		CASE pMzTool^.P_eObjectType OF
			E_ObjectType.OBJECTTYPE_CartDispenser,
			E_ObjectType.OBJECTTYPE_CartDispStirrer,
			E_ObjectType.OBJECTTYPE_MultiCartHolder,
			E_ObjectType.OBJECTTYPE_PassivPip,
			E_ObjectType.OBJECTTYPE_PiezoPip,
			E_ObjectType.OBJECTTYPE_SolenoidPip,
			E_ObjectType.OBJECTTYPE_PowderPip,
			E_ObjectType.OBJECTTYPE_Extruder,
			E_ObjectType.OBJECTTYPE_TwinExtruder,
			E_ObjectType.OBJECTTYPE_Luer,
			E_ObjectType.OBJECTTYPE_TitrationTool,
			E_ObjectType.OBJECTTYPE_PickPlacePip:
				bMeasureTip := TRUE;
			E_ObjectType.OBJECTTYPE_HybridDispenser:
				//Gemessen wird mit dem MasterTool des Dispensers
				pHybridDispenser := pMzTool;
				pMzTool := pHybridDispenser^.P_pMasterTool;
				bMeasureTip := TRUE;
			E_ObjectType.OBJECTTYPE_StampSupport:	//Vermessung Stamp
				pStampSupport := fbObjectDirectory.M_GetObjPointer(refActionData.nObject);
				IF fbObjectDirectory.M_GetObjType(refActionData.nTarget) = E_ObjectType.OBJECTTYPE_InkStation THEN
					pInkStation := pTarget;
					iTargetZSensor := pInkStation^;
				ELSIF fbObjectDirectory.M_GetObjType(refActionData.nTarget) = E_ObjectType.OBJECTTYPE_StampMagazine THEN
					pStampMagazine := pTarget; 
					iTargetZSensor := pStampMagazine^;
				END_IF
				IF iTargetZSensor.P_bSensor THEN
					M_ExeAction := E_ErrorIdCmd.ERRORID_SensorAlreadySwitched;
					RETURN;
				END_IF
				bMeasureStamp := TRUE;
			E_ObjectType.OBJECTTYPE_ZSensor:	//Vermessung Target
				IF eMeasTipOption = E_MeasureOption.MEAS_OPTION_SlowApproach OR eMeasTipOption = E_MeasureOption.MEAS_OPTION_FastApproach THEN
					bMeasureTarget := TRUE;
				ELSE
					M_ExeAction := E_ErrorIdCmd.ERRORID_InvalidMeasureOption;
					RETURN;				
				END_IF
			ELSE
				M_ExeAction := E_ErrorIdCmd.ERRORID_UnsuitableObject; //Error
				RETURN;				
		END_CASE
		
		
		//Wenn bMeasureTip, dann muss Target ein TipCalibrator sein
		IF bMeasureTip OR bCalibrateTipCalibrator THEN
			IF NOT pTarget^.P_eObjectType = E_ObjectType.OBJECTTYPE_TipCalibrator THEN
				bMeasureTip := FALSE;
				bCalibrateTipCalibrator := FALSE;
				M_ExeAction := E_ErrorIdCmd.ERRORID_UnsuitableTarget;  //Error
				RETURN;
			END_IF
			pTipCalibrator := pTarget;
			bMeasureTipLegacy := pTipCalibrator^.P_bLegacy;
			
			IF pMzTool^.P_pPiece = 0 THEN
				IF pMzTool^.P_eObjectType = E_ObjectType.OBJECTTYPE_PassivPip OR
				   pMzTool^.P_eObjectType = E_ObjectType.OBJECTTYPE_PiezoPip OR
				   pMzTool^.P_eObjectType = E_ObjectType.OBJECTTYPE_SolenoidPip OR
				   pMzTool^.P_eObjectType = E_ObjectType.OBJECTTYPE_Luer THEN
				   rMeasureDistance := 6000;
				ELSIF pMzTool^.P_eObjectType = E_ObjectType.OBJECTTYPE_TitrationTool THEN 
				   rMeasureDistance := 10000;
				ELSE
					M_ExeAction := E_ErrorIdCmd.ERRORID_NoPieceOnTool;
					RETURN;
				END_IF
			ELSE
				IF NOT(pMzTool^.P_pPiece^.P_eObjectType = E_ObjectType.OBJECTTYPE_Nozzle OR
					pMzTool^.P_pPiece^.P_eObjectType = E_ObjectType.OBJECTTYPE_Needle OR
					pMzTool^.P_pPiece^.P_eObjectType = E_ObjectType.OBJECTTYPE_Tip) THEN
					M_ExeAction := E_ErrorIdCmd.ERRORID_InvalidPieceType;
					RETURN;
				ELSE
					rMeasureDistance := pMzTool^.P_pPiece^.P_rMeasureDistance;
				END_IF
			END_IF
		END_IF
		
		M_ExeAction := pMzTool^.M_CheckAction(refActionData, pTarget); //Action mit MzTool ausführbar?
		IF M_ExeAction > 0 THEN
			bMeasureTip := FALSE;
			RETURN;
		END_IF
		
		pHighVoltTray := pTarget^.M_GetFirstParentOfType(E_ObjectType.OBJECTTYPE_HighVoltTray);
		IF pHighVoltTray > 0 THEN
			IF pHighVoltTray^.P_nCurrentVoltage > cHighVoltThreshold THEN //>20 da anloger Eingang etwas rauscht
				M_ExeAction := E_ErrorIdCmd.ERRORID_RiskHighvoltFlashover;
				RETURN;
			END_IF
		END_IF
		
		
	E_Action.ACTION_MoveAllHome:
		;

	E_Action.ACTION_MoveToTarget:
		//Tool ermitteln
		IF fbObjectDirectory.M_ObjIsMzTool(refActionData.nObject) THEN //Gültiges MzTool?
			pMzTool := fbObjectDirectory.M_GetObjPointer(refActionData.nObject);
		ELSE 
			M_ExeAction := E_ErrorIdCmd.ERRORID_UnsuitableObject;  //Error
			RETURN;
		END_IF
		
		IF NOT (fbObjectDirectory.M_GetObjType(refActionData.nObject) = E_ObjectType.OBJECTTYPE_MZHead) THEN
			M_ExeAction := pMzTool^.M_AskSiblingForAction(E_Action.ACTION_MoveToTarget);
			IF M_ExeAction > 0 THEN
				RETURN;
			END_IF
		END_IF
		
		//Falls das Target sich auf dem HighVoltTray befindet und dieses auch angeschalten ist, dann ist ein MoveToTarget nur
		//mit einem MES-Tool möglich
		pTarget := fbObjectDirectory.M_GetObjPointer(refActionData.nTarget);
		IF pTarget = 0 THEN
			M_ExeAction := E_ErrorIdCmd.ERRORID_UnsuitableObject;  //Error
		END_IF
		pHighVoltTray := pTarget^.M_GetFirstParentOfType(E_ObjectType.OBJECTTYPE_HighVoltTray);
		IF pHighVoltTray > 0 THEN
			IF pHighVoltTray^.P_nCurrentVoltage > cHighVoltThreshold AND NOT pMzTool^.P_bIsMESTool THEN
				M_ExeAction := E_ErrorIdCmd.ERRORID_RiskHighvoltFlashover;
				RETURN;
			END_IF
		END_IF
	
		M_ExeAction := fbMoveToTarget.M_SetAndCheckParams(refActionData);

		IF M_ExeAction > 0 THEN
			RETURN;
		END_IF
		
	E_Action.ACTION_OpenCloseFlipTube:
		IF fbObjectDirectory.M_ObjIsMzTool(refActionData.nObject) THEN //Gültiges MzTool?
			pMzTool := fbObjectDirectory.M_GetObjPointer(refActionData.nObject);
		ELSE 
			M_ExeAction := E_ErrorIdCmd.ERRORID_UnsuitableObject;  //Error
			RETURN;
		END_IF
		
		IF fbObjectDirectory.M_ObjIsTarget(refActionData.nTarget) THEN //Gültiges Target?
			pTarget := fbObjectDirectory.M_GetObjPointer(refActionData.nTarget);
			IF pTarget^.P_eObjectType = E_ObjectType.OBJECTTYPE_FlipTubeRack THEN //Target ein FlipTubeRack?
				pFlipTubeRack := pTarget;
				pPieceSlot := pFlipTubeRack^.M_GetSlot(DINT_TO_UINT(refActionData.aParams[1]));
			ELSE
				M_ExeAction := E_ErrorIdCmd.ERRORID_UnsuitableTarget;  //Error	
			END_IF
		ELSE
			M_ExeAction := E_ErrorIdCmd.ERRORID_UnsuitableTarget;  //Error
			RETURN;
		END_IF
		
		M_ExeAction := pMzTool^.M_CheckAction(refActionData, pTarget); //Ausführbar mit Target?
		IF M_ExeAction > 0 THEN
			RETURN;
		END_IF
		
		M_ExeAction := pTarget^.M_CheckAction(refActionData, pMzTool); //Ausführbar mit MzTool?
		IF M_ExeAction > 0 THEN
			RETURN;
		END_IF
		bOpen := NOT DINT_TO_BOOL(refActionData.aParams[2]); //Öffen
		
	E_Action.ACTION_StampDemolding:
		IF fbObjectDirectory.M_GetObjType(refActionData.nObject) <> E_ObjectType.OBJECTTYPE_StampSupport THEN //Gültiges MzTool?
			M_ExeAction := E_ErrorIdCmd.ERRORID_UnsuitableObject;
			RETURN;
		END_IF
		pMzTool := fbObjectDirectory.M_GetObjPointer(refActionData.nObject);
		pStampSupport := pMzTool;

		M_ExeAction := pStampSupport^.M_CheckAction(refActionData,0);
		IF M_ExeAction > 0 THEN
			RETURN;
		END_IF
 
		nDistance1 := refActionData.aParams[1];
		nSpeed1 := refActionData.aParams[2];
		nPressure1 := DINT_TO_INT(refActionData.aParams[3]);
		nPressure2 := DINT_TO_INT(refActionData.aParams[4]);
		nPeriode := refActionData.aParams[5];
		nDutycycle := refActionData.aParams[6];
		
	E_Action.ACTION_StampInking:
		IF fbObjectDirectory.M_GetObjType(refActionData.nObject) <> E_ObjectType.OBJECTTYPE_StampSupport THEN //Gültiges MzTool?
			M_ExeAction := E_ErrorIdCmd.ERRORID_UnsuitableObject;
			RETURN;
		END_IF
		
		//Inking kann an einem Punkt oder an der InkStation stattfinden
		IF fbObjectDirectory.M_GetObjType(refActionData.nTarget) = E_ObjectType.OBJECTTYPE_InkStation THEN
			pInkStation := fbObjectDirectory.M_GetObjPointer(refActionData.nTarget);
		ELSIF fbObjectDirectory.M_GetObjType(refActionData.nTarget) = E_ObjectType.OBJECTTYPE_Point THEN
			pInkStation := 0;
		ELSE
			M_ExeAction := E_ErrorIdCmd.ERRORID_UnsuitableTarget;
			RETURN;
		END_IF
		
		//Wozu brauchen wir hier das Target?
		pTarget := fbObjectDirectory.M_GetObjPointer(refActionData.nTarget);
		pStampSupport := fbObjectDirectory.M_GetObjPointer(refActionData.nObject);
		
		M_ExeAction := pStampSupport^.M_CheckAction(refActionData,pTarget);
		IF M_ExeAction > 0 THEN
			RETURN;
		END_IF
		
		nDistance1 := refActionData.aParams[1];
		nPressure1 := DINT_TO_INT(refActionData.aParams[2]);
		nTime := DINT_TO_DWORD(refActionData.aParams[3]);
		
	E_Action.ACTION_TeachTarget:
		//Object gültig?
		IF NOT fbObjectDirectory.M_ObjIsMzTool(refActionData.nObject) THEN
			M_ExeAction := E_ErrorIdCmd.ERRORID_UnsuitableObject;  //Error
			RETURN;
		END_IF
		
		IF fbObjectDirectory.M_ObjIsTarget(refActionData.nTarget) THEN
			pTarget := fbObjectDirectory.M_GetObjPointer(refActionData.nTarget);
			IF pTarget > 0 THEN
				M_ExeAction := pTarget^.M_CheckAction(refActionData, pMzTool);
				IF M_ExeAction > 0 THEN
					RETURN;
				END_IF
			ELSE
				M_ExeAction := E_ErrorIdCmd.ERRORID_UnsuitableTarget;  //Error
				RETURN;
			END_IF
		ELSE
			M_ExeAction := E_ErrorIdCmd.ERRORID_UnsuitableTarget;  //Error
			RETURN;
		END_IF
		//Target gültig? (derzeit nur Mtp impl.)
		
		//Hier macht es Sinn, beim Target selber zu fragen, ob es sich einteachen lässt
		
		(*IF fbObjectDirectory.M_GetObjType(refActionData.nTarget) = E_ObjectType.OBJECTTYPE_Mtp THEN
			pMtp := aI_Object[refActionData.nTarget].P_pObject;
		ELSIF fbObjectDirectory.M_GetObjType(refActionData.nTarget) = E_ObjectType.OBJECTTYPE_Point THEN
			;
		ELSIF fbObjectDirectory.M_GetObjType(refActionData.nTarget) = E_ObjectType.OBJECTTYPE_Stroboscope THEN
			;
		ELSE
			M_ExeAction := E_ErrorIdCmd.ERRORID_InvalidTarget;  //Error
			RETURN;
		END_IF*)
		
		pMzTool := fbObjectDirectory.M_GetObjPointer(refActionData.nObject);
		pTarget := fbObjectDirectory.M_GetObjPointer(refActionData.nTarget);
		IF pTarget^.P_eObjectType = E_ObjectType.OBJECTTYPE_Mtp THEN
			pMtp := pTarget;
		END_IF
		eTargetRef := DINT_TO_USINT(refActionData.aParams[1]);
		nSpecPointSlotNr := DINT_TO_UINT(refActionData.aParams[2]);
		nZOffset1 := refActionData.aParams[3];
		//refActionData.aParams[4] ist Reserve
		eTeachOption := DINT_TO_USINT(refActionData.aParams[5]);
		
		pHighVoltTray := pTarget^.M_GetFirstParentOfType(E_ObjectType.OBJECTTYPE_HighVoltTray);
		IF pHighVoltTray > 0 THEN
			IF pHighVoltTray^.P_nCurrentVoltage > cHighVoltThreshold THEN
				M_ExeAction := E_ErrorIdCmd.ERRORID_RiskHighvoltFlashover;
				RETURN;
			END_IF
		END_IF
		
	E_Action.ACTION_TeachTool:
		IF NOT fbObjectDirectory.M_ObjIsMzTool(refActionData.nObject) THEN
			M_ExeAction := E_ErrorIdCmd.ERRORID_UnsuitableObject;  //Error
			RETURN;
		END_IF
		//Target gültig?
		IF NOT fbObjectDirectory.M_ObjIsTarget(refActionData.nTarget) THEN
			M_ExeAction := E_ErrorIdCmd.ERRORID_UnsuitableTarget;  //Error
			RETURN;
		END_IF
		pMzTool := fbObjectDirectory.M_GetObjPointer(refActionData.nObject);
		pTarget := fbObjectDirectory.M_GetObjPointer(refActionData.nTarget);
		eTargetRef := DINT_TO_USINT(refActionData.aParams[1]);
		nCol := DINT_TO_USINT(refActionData.aParams[2]);
		nRow := DINT_TO_USINT(refActionData.aParams[2]);
		nZOffset1 := refActionData.aParams[4];

		pHighVoltTray := pTarget^.M_GetFirstParentOfType(E_ObjectType.OBJECTTYPE_HighVoltTray);
		IF pHighVoltTray > 0 THEN
			IF pHighVoltTray^.P_nCurrentVoltage > cHighVoltThreshold THEN
				M_ExeAction := E_ErrorIdCmd.ERRORID_RiskHighvoltFlashover;
				RETURN;
			END_IF
		END_IF

	E_Action.ACTION_TransferGas:
		//Beteiligte Luers checken
		IF NOT fbObjectDirectory.M_GetObjType(refActionData.nObject) = E_ObjectType.OBJECTTYPE_Luer THEN
			M_ExeAction := E_ErrorIdCmd.ERRORID_UnsuitableObject;  //Error
			RETURN;
		END_IF

		IF NOT fbObjectDirectory.M_GetObjType(refActionData.nTarget) = E_ObjectType.OBJECTTYPE_Luer THEN
			M_ExeAction := E_ErrorIdCmd.ERRORID_UnsuitableObject;  //Error
			RETURN;
		END_IF
		pLuer := fbObjectDirectory.M_GetObjPointer(refActionData.nObject);
		pLuer2 := fbObjectDirectory.M_GetObjPointer(refActionData.nTarget);
		nPressure1 := DINT_TO_INT(refActionData.aParams[1]);
		nTime := DINT_TO_DWORD(refActionData.aParams[2]);
		
	E_Action.ACTION_TransferLiquid:
		//Beteiligte Luers checken
		IF NOT fbObjectDirectory.M_GetObjType(refActionData.nObject) = E_ObjectType.OBJECTTYPE_Luer THEN
			M_ExeAction := E_ErrorIdCmd.ERRORID_UnsuitableObject;  //Error
			RETURN;
		END_IF

		IF NOT fbObjectDirectory.M_GetObjType(refActionData.nTarget) = E_ObjectType.OBJECTTYPE_Luer THEN
			M_ExeAction := E_ErrorIdCmd.ERRORID_UnsuitableTarget;  //Error
			RETURN;
		END_IF
		pLuer := fbObjectDirectory.M_GetObjPointer(refActionData.nObject);
		pLuer2 := fbObjectDirectory.M_GetObjPointer(refActionData.nTarget);
		pDiluter1 := pLuer^.P_pDiluter;
		pDiluter2 := pLuer2^.P_pDiluter;
		
		nQuantity1 := refActionData.aParams[1];
		nFlow1 := refActionData.aParams[2];
		nQuantity2 := refActionData.aParams[3];
		nQuantity3 := refActionData.aParams[4];
		
	E_Action.ACTION_TransferTray:
		//Hier schon Bedingungen abfragen.
		IF fbObjectDirectory.M_GetObjType(refActionData.nObject) = E_ObjectType.OBJECTTYPE_TrayTransporter THEN
			pTrayTransporter := fbObjectDirectory.M_GetObjPointer(refActionData.nObject);
		ELSE
			M_ExeAction := E_ErrorIdCmd.ERRORID_UnsuitableObject;  //Error
			RETURN;
		END_IF
 
		eTransferTrayCtrl :=  DINT_TO_USINT(refActionData.aParams[1]);

	E_Action.ACTION_WashTool:
		IF fbObjectDirectory.M_ObjIsMzTool(refActionData.nObject) THEN //Gültiges MzTool?
			pMzTool := fbObjectDirectory.M_GetObjPointer(refActionData.nObject);
		ELSE 
			M_ExeAction := E_ErrorIdCmd.ERRORID_UnsuitableObject;  //Error
			RETURN;
		END_IF	
		
		IF fbObjectDirectory.M_GetObjType(refActionData.nTarget) <> E_ObjectType.OBJECTTYPE_WashStation THEN //gültiges Target?
			M_ExeAction := E_ErrorIdCmd.ERRORID_UnsuitableTarget;
			RETURN;
		ELSE
			pTarget := fbObjectDirectory.M_GetObjPointer(refActionData.nTarget);
			pWashStation := pTarget;
		END_IF
		
		//Kann Tool Action ausführen?
		M_ExeAction := pMzTool^.M_CheckAction(refActionData, pTarget);
		IF M_ExeAction > 0 THEN
			RETURN;
		END_IF
		
		//Kann WashStation Action ausführen?
		M_ExeAction := pWashStation^.M_CheckAction(refActionData, pMzTool);
		IF M_ExeAction > 0 THEN
			RETURN;
		END_IF
		
		nSpecPointSlotNr := DINT_TO_UINT(refActionData.aParams[1]);
		//RinseChannel aus WashStation holen
		nRinseChannel := pWashStation^.M_GetRinseChannel(UINT_TO_USINT(nSpecPointSlotNr));
		eWashMode := DINT_TO_USINT(refActionData.aParams[2]);
		//passt WashMode zu RinseChannel?
		IF (eWashMode = E_WashMode.MODE_WashInOutside) OR (eWashMode = E_WashMode.MODE_WashOutside) THEN
			IF nRinseChannel = 0 THEN
				M_ExeAction := E_ErrorIdCmd.ERRORID_InvalidRinseChannel;
				RETURN;
			END_IF
		END_IF
		
		nQuantity1 := refActionData.aParams[3];
		nFlow1 := refActionData.aParams[4];
		nTime := DINT_TO_DWORD(refActionData.aParams[5]);
		nDilInputNr := refActionData.aParams[6];

 	ELSE
		M_ExeAction := E_ErrorIdCmd.ERRORID_InvalidAction; //Error		
END_CASE
bBusy := TRUE;
eCurrentAction := refActionData.eAction;
eCurrentState := E_MachineState.MACHINESTATE_Active;
END_METHOD

METHOD M_Pause
VAR_INPUT
END_VAR
//derzeit wird nur DispenseTest in Pause versetzt
IF eCurrentState = E_MachineState.MACHINESTATE_Active THEN
	IF eCurrentAction = E_Action.ACTION_DispenseTest THEN
		eCurrentState := E_MachineState.MACHINESTATE_PauseRequest;
	END_IF
END_IF
END_METHOD

METHOD M_Reset
VAR_INPUT
END_VAR
VAR
END_VAR
IF eCurrentState = E_MachineState.MACHINESTATE_Error THEN
	bBusy := TRUE;
	eCurrentState := E_MachineState.MACHINESTATE_Reset;
END_IF
END_METHOD

METHOD M_Stop
VAR_INPUT
END_VAR
IF eCurrentState = E_MachineState.MACHINESTATE_Active OR 
	eCurrentState = E_MachineState.MACHINESTATE_PauseRequest OR
	eCurrentState = E_MachineState.MACHINESTATE_Pause THEN
	
	bStop := TRUE;
END_IF
END_METHOD

METHOD M_StopAction
VAR_INPUT
	eAction : E_Action;
END_VAR
IF eCurrentAction = eAction THEN
	M_Stop();
END_IF
END_METHOD

PROPERTY P_bLastActionResult : BOOL
GET
P_bLastActionResult := bLastActionResult;
END_GET
SET
bLastActionResult := P_bLastActionResult;
END_SET
END_PROPERTY

PROPERTY P_bPauseRequestIntern : BOOL
GET
P_bPauseRequestIntern := bPauseRequestIntern;
END_GET
SET
bPauseRequestIntern := P_bPauseRequestIntern;
END_SET
END_PROPERTY

PROPERTY P_nDispenseTrials : DINT
GET
P_nDispenseTrials := nDispenseTrials;
END_GET
SET
nDispenseTrials := P_nDispenseTrials;
END_SET
END_PROPERTY

PROPERTY P_nLastActionResult : DINT
GET
P_nLastActionResult := nLastActionResult;
END_GET
SET
nLastActionResult := P_nLastActionResult;
END_SET
END_PROPERTY

END_FUNCTION_BLOCK

// ---- Hardware/MultiZ/FB_ZM_ReadZSensorID.TcPOU
FUNCTION_BLOCK FB_ZM_ReadZSensorID
VAR_INPUT
	bExecute		: BOOL;
	pFbZAxisRef		: POINTER TO FB_ZAxisRef;
END_VAR
VAR_OUTPUT
	bBusy			: BOOL;
	bCommandAborted	: BOOL;
	bError			: BOOL;
	nErrorID		: ERRORID;	
END_VAR
VAR
	nState				: USINT;
	timeOut				: TON;
	fbSdoRead			: FB_SDO_READ;
END_VAR

//Die Id (eigentlich der Offset) wird ausgelesen, indem eine kurze Vermessung mit 100µm Distanz gestartet wird.
//Als Ergebnis bringt die Achse einen der 3 folgenden Fehler:
//1. No_Z-Limit -> kein ZSensor (Id wurde nicht ausgelesen)
//2. Z_Limit_Fail -> ZSensor betätigt (Id wurde ausgelesen)
//3. Z_Limit_not_found -> (Id wurde ausgelesen)

IF bExecute THEN
	IF pFbZAxisRef = 0 THEN
		nErrorId := E_ErrorIdMultiZ.ERRORID_InvalidZChannel;
		bBusy := FALSE;
		bError := TRUE;
		nState := 99;
		RETURN;
	END_IF

	//Wenn durch anderen FB Achse gestoppt, dann abbrechen
	IF pFbZAxisRef^.stStatus.bCmdAborted THEN //Muss noch irgendwo gesetzt werden!!!!
		bCommandAborted := TRUE;
		bBusy := FALSE;
	END_IF
	
	timeOut();
	IF timeOut.Q THEN
		bBusy := FALSE;
		bError := TRUE;
		nState := 99;
		RETURN;
	END_IF

	CASE nState OF
		0: 	//Nur folgende Tools können ZSensor aufnehmen
			bBusy := TRUE;
			IF NOT (pFbZAxisRef^.eFixedToolType = E_MzToolType.TOOL_TYPE_PiezoPip OR 
					pFbZAxisRef^.eFixedToolType = E_MzToolType.TOOL_TYPE_PiezoSingle OR 
					pFbZAxisRef^.eFixedToolType = E_MzToolType.TOOL_TYPE_SyringeExtruder) THEN
				nErrorID := E_ErrorIdCmd.ERRORID_ConfigErrorZSensor;
				bBusy := FALSE;
				bError := TRUE;
				nState := 99;
				RETURN;
			END_IF
			
			pFbZAxisRef^.stStatus.bIsMoving := TRUE;
			pFbZAxisRef^.stStatus.bHasJob := TRUE;
        	//Geschwindigkeit setzen
			pFbZAxisRef^.stOutput.nVelo := REAL_TO_DINT(pFbZAxisRef^.P_rMaxSpeed);
			//Aktuelle Position ? Wenn ganz unten steht, dann 200µ nach oben fahren
			IF (pFbZAxisRef^.P_rCurrentPos - 100.0) < pFbZAxisRef^.P_rMinPos THEN
				//200µm nach oben fahren
				pFbZAxisRef^.stOutput.nMode := 1; //normaler Positioniermodus
				pFbZAxisRef^.P_rAbsTargetPos := pFbZAxisRef^.P_rMinPos + 200.0;
				pFbZAxisRef^.stOutput.nCtrl := 1;
				nState := 1;
			ELSE
				nState := 3;
			END_IF
			
		1:	//SetpointAcknowledge?
			IF pFbZAxisRef^.stInput.nStatus.1 THEN
				pFbZAxisRef^.stOutput.nCtrl.0 := FALSE;	//Fahrauftrag zurücksetzen
				timeOut(IN:= FALSE);
				nState := 2;
			ELSE
				timeOut(IN:= TRUE, PT:=T#1000MS);	//Timer für Timeout starten
			END_IF
			
		2:  //TargetReached?
			IF pFbZAxisRef^.stInput.nStatus.0 THEN
				timeOut(IN:= FALSE);
				nState := 3;
			ELSE
				timeOut(IN:= TRUE, PT:= T#1000MS);	//Timer für Timeout starten
			END_IF			
			
		3:	//100µm nach unten im Messmodus fahren -> sollte in jedem Fall einen Fehler erzeugen
			//Hier muss kurzzeitig verhindert werden, dass dieser Fehler in Action "A_Monitor" von
			//FB_MultiZRef abgefangen wird
			pFbZAxisRef^.stOutput.nMode := 5; //normaler Messmodus
			pFbZAxisRef^.stOutput.nTrgtPos := 100;
			pFbZAxisRef^.bIngoreError := TRUE;
			nState := 4;
			
		4:	pFbZAxisRef^.stOutput.nCtrl := 1;
			nState := 5;
			
		5:	//SetpointAcknowledge?
			IF pFbZAxisRef^.stInput.nStatus.1 THEN
				pFbZAxisRef^.stOutput.nCtrl.0 := FALSE;	//Fahrauftrag zurücksetzen
				timeOut(IN:= FALSE);
				timeOut(IN:= TRUE, PT:= T#1S);
				nState := 6;
			ELSE
				timeOut(IN:= TRUE, PT:=T#1000MS);	//Timer für Timeout starten
			END_IF

		6:	//Hier sollte jetzt ein Fehler kommen
			IF pFbZAxisRef^.stInput.nStatus.3 AND pFbZAxisRef^.stInput.nError > 0 THEN
				pFbZAxisRef^.stOutput.nMode := 0; //Mode muss zum Zurücksetzen des Fehlers auf 0 sein
				timeOut(IN:= FALSE);
				nErrorID := pFbZAxisRef^.stInput.nError;
				IF nErrorID = 19 OR nErrorID = 20 THEN
					//weiter zu Offset auslesen und Error zurücksetzen
					fbSdoRead(sADSNetID:= pFbZAxisRef^.pMultiZRef^.P_sAdsNetId,	nPortNr:= pFbZAxisRef^.pMultiZRef^.P_nAdsPort,
							nIndex:= cZSensOffset.nIndex, nSubIndex:= pFbZAxisRef^.nChannel, nDataLength:= cZSensOffset.nLength, bExecute:= TRUE);					
					nState := 7;
				ELSE
					nErrorID := F_MultiZError_TO_ErrorId(pFbZAxisRef^.stInput.nError);
					bBusy := FALSE;
					bError := TRUE;
					RETURN;					
				END_IF
			END_IF
			
		7:	//Warten bis ZOffset ausgelesen
			fbSdoRead();
			IF NOT fbSdoRead.bBusy THEN
				IF fbSdoRead.bError THEN
					nErrorID := fbSdoRead.nAdsErrorId;
					bError := TRUE;
					nState := 99;
				ELSE
					nState := 8;
					pFbZAxisRef^.stOutput.nCtrl := 8;	//Error zurücksetzen
					pFbZAxisRef^.P_nZSensorID := fbSdoRead.nData;
				END_IF
				fbSdoRead(bExecute:= FALSE);
			END_IF
			
		8:	IF NOT pFbZAxisRef^.stInput.nStatus.3 AND pFbZAxisRef^.stInput.nError = 0 THEN
				pFbZAxisRef^.stOutput.nCtrl := 0;
				bBusy := FALSE;				
			END_IF
	END_CASE
ELSE
	bBusy := FALSE;
	nState := 0;
	bError := FALSE;
	nErrorID := 0;
	timeOut(IN:=FALSE);
	pFbZAxisRef^.stStatus.bCmdAborted := FALSE;
	pFbZAxisRef^.stOutput.nMode := 0;
	pFbZAxisRef^.stStatus.bHasJob := FALSE;
	pFbZAxisRef^.stStatus.bIsMoving := FALSE;
	pFbZAxisRef^.bIngoreError := FALSE;
END_IF

END_FUNCTION_BLOCK

// ---- Actions/FB_MeasTip.TcPOU
FUNCTION_BLOCK FB_MeasTip
VAR_INPUT
	bExecute 		: BOOL;
	pMzTool			: POINTER TO FB_MzBase;
	pTipCalibrator	: POINTER TO FB_TipCalibrator;
	nDirection 		: USINT;	//1: X, 2: Y, 3: Z
	nZFeedStart		: DINT;		//Anfangsschrittweite in Z (µm)
	nZFeedEnde		: DINT;		//Endschrittweite in Z (µm)
	nZFeedMax		: DINT;
	stStartPos		: ST_3DPoint;
	stEndPos		: ST_3DPoint;
	stTempPoint		: ST_3DPoint;
END_VAR
VAR_OUTPUT
	bBusy		: BOOL;
	bError		: BOOL;
	nErrorId	: ERRORID;
	stProbePos	: ST_3DPoint;
END_VAR
VAR
	stError				: ST_Error;
	pXDrive				: POINTER TO FB_XYDriveBase;
	pYDrive				: POINTER TO FB_XYDriveBase;
	nState				: USINT;
	stCurrentPos		: ST_3DPoint;
	stCalibPoint		: ST_3DPoint;
	stPassIntersect		: ST_3DPoint;	
	stActionData		: ST_ActionData;
	rCapturedPos1		: REAL;
	rCapturedPos2		: REAL;
	nStateA_ProbeX		: USINT;
	nStateA_ProbeY		: USINT;
	bSingleProbe		: BOOL;
	bDirPositive		: BOOL;
	nStartPos			: DINT;
	nEndPos				: DINT;
	bBeginStartPos		: BOOL;
	nProbeSpeed			: DINT := 20000;
	bProbeSuccess		: BOOL;
	nProbeErrorId		: UINT;
	bProbePositiveOK	: BOOL;
	bProbeNegativeOK	: BOOL;
	bProbeMissingTouch	: BOOL;
	bProbeFlag			: BOOL;
	bTouchProbe			: BOOL;
	nProbeCount			: USINT;
	nZFeed				: DINT;
	nZFeedSum			: DINT;
	bMaxFeedAchieved	: BOOL;
END_VAR

IF bExecute THEN
	IF nDirection = 1 THEN	//X
		A_MeasureX();
	ELSIF nDirection = 2 THEN //Y
		A_MeasureY();
	ELSIF nDirection = 3 THEN	//Z
		A_MeasureZ();
	END_IF
ELSE
	bError := FALSE;
	nErrorId := 0;
	nState := 0;
	nStateA_ProbeX := 0;
	nStateA_ProbeY := 0;
END_IF

ACTION A_MeasureX:
IF pMzTool^.P_bError THEN
	nState := 99;
	bError := TRUE;
	stError := pMzTool^.P_stError;
	nErrorId := stError.ErrorId; 
END_IF

CASE nState OF
	0:	
		nStartPos := REAL_TO_DINT(stStartPos.X);
		nEndPos := REAL_TO_DINT(stEndPos.X);
		bBusy := TRUE;
		bBeginStartPos := TRUE;
		bSingleProbe := FALSE;
		nState := 1;

	1:	//XProbe
		A_ProbeX();
		IF nStateA_ProbeX = 80 THEN
			nStateA_ProbeX := 0;
			IF bProbeSuccess AND bProbePositiveOK AND bProbeNegativeOK THEN
				//Checken, ob beide Probe-Positionen nicht zu weit voneinander abweichen (max5mm)
				IF ABS(rCapturedPos1 - rCapturedPos2) > 20000 THEN
					bError := TRUE;
					nErrorId := E_ErrorIdCmd.ERRORID_MeasureTouchProbeFail;
					bBusy := FALSE;
					RETURN;	
				END_IF				
				stTempPoint.X := (rCapturedPos1 + rCapturedPos2) / 2;
				stTempPoint :=  pMzTool^.M_RawPosToRealPos(stTempPoint);
				stProbePos.X := stTempPoint.X;
				bBusy := FALSE;	
			END_IF
		ELSIF nStateA_ProbeX = 99 THEN
			nStateA_ProbeX := 0;
			bBusy := FALSE;
			bError := TRUE;
			nErrorId := nProbeErrorId;
		END_IF
		
	70:	//Abbrechen
		IF nStateA_ProbeX > 0 THEN
			nStateA_ProbeX := 70;
			A_ProbeX();
			nState := 71;
		END_IF
		
	71:	
		A_ProbeX();
		IF nStateA_ProbeX >= 80 THEN
			IF nStateA_ProbeX >= 99 THEN
				nErrorId := nProbeErrorId;
				bError := TRUE;
			END_IF
			nStateA_ProbeX := 0;
			bBusy := FALSE;
		END_IF
END_CASE
END_ACTION

ACTION A_MeasureY:
IF pMzTool^.P_bError THEN
	nState := 90;
	bError := TRUE;
	stError := pMzTool^.P_stError;
	nErrorId := stError.ErrorId; 
END_IF

CASE nState OF
	0:	
		nStartPos := REAL_TO_DINT(stStartPos.Y);
		nEndPos := REAL_TO_DINT(stEndPos.Y);
		bBusy := TRUE;
		bBeginStartPos := FALSE;
		bSingleProbe := FALSE;
		nState := 1;

	1:	//YProbe
		A_ProbeY();
		IF nStateA_ProbeY = 80 THEN
			nStateA_ProbeY := 0;
			IF bProbeSuccess AND bProbePositiveOK AND bProbeNegativeOK THEN
				//Checken, ob beide Probe-Positionen nicht zu weit voneinander abweichen (max5mm)
				IF ABS(rCapturedPos1 - rCapturedPos2) > 20000 THEN
					bError := TRUE;
					nErrorId := E_ErrorIdCmd.ERRORID_MeasureTouchProbeFail;
					bBusy := FALSE;
					RETURN;	
				END_IF
				stTempPoint.Y := (rCapturedPos1 + rCapturedPos2) / 2;
				stTempPoint :=  pMzTool^.M_RawPosToRealPos(stTempPoint);
				stProbePos.Y := stTempPoint.Y;
				bBusy := FALSE;	
			END_IF
		ELSIF nStateA_ProbeY = 99 THEN
			nStateA_ProbeY := 0;
			bBusy := FALSE;
			bError := TRUE;
			nErrorId := nProbeErrorId;
		END_IF
		
	70:	//Abbrechen
		IF nStateA_ProbeY > 0 THEN
			nStateA_ProbeY := 70;
			A_ProbeY();
			nState := 71;
		END_IF
		
	71:	
		A_ProbeY();
		IF nStateA_ProbeY >= 80 THEN
			IF nStateA_ProbeY >= 99 THEN
				bError := TRUE;
			END_IF
			nStateA_ProbeY := 0;
			bBusy := FALSE;
		END_IF		
END_CASE
END_ACTION

ACTION A_MeasureZ:
IF pMzTool^.P_bError THEN
	nState := 90;
	stError := pMzTool^.P_stError;
	nErrorId := stError.ErrorId; 
END_IF
		
CASE nState OF
	0:	//
		nStartPos := REAL_TO_DINT(stStartPos.X);
		nEndPos := REAL_TO_DINT(stEndPos.X);
		nZFeed := nZFeedStart;
		bBusy := TRUE;
		nZFeedSum := 0;
		bBeginStartPos := TRUE;
		bMaxFeedAchieved := FALSE;
		nState := 1;

	1:	//XProbe
		bSingleProbe := TRUE;
		IF nZFeed > 0 THEN
			bProbeMissingTouch := TRUE;
		ELSE
			bProbeMissingTouch := FALSE;
		END_IF
		
		A_ProbeX();
		IF nStateA_ProbeX = 80 THEN
			nStateA_ProbeX := 0;
			bBeginStartPos := FALSE;
			IF bProbeSuccess THEN
				//wenn hier schon erfolgreich, dann noch einmal in die andere Richtung und dann auf Encoderwert fahren
				IF bProbePositiveOK XOR bProbeNegativeOK THEN
					RETURN;
				ELSIF bProbePositiveOK AND bProbeNegativeOK THEN
					//Checken, ob beide Probe-Positionen nicht zu weit voneinander abweichen (max5mm)
					IF ABS(rCapturedPos1 - rCapturedPos2) > 20000 THEN
						bError := TRUE;
						nErrorId := E_ErrorIdCmd.ERRORID_MeasureTouchProbeFail;
						bBusy := FALSE;
						RETURN;	
					END_IF					
					//auf ermittelten Wert fahren
					nState := 4;
				ELSE
					bError := TRUE;
					bBusy := FALSE;
				END_IF
			ELSE
				nState := 2;
			END_IF
			
		ELSIF nStateA_ProbeX = 99 THEN
			nStateA_ProbeX := 0;
			bBusy := FALSE;
			nErrorId := nProbeErrorId;
			bError := TRUE;
		END_IF
		
	2:	//ZMove
		IF bMaxFeedAchieved THEN
			bError := TRUE;
			nErrorId := E_ErrorIdCmd.ERRORID_MeasureZDistanceExeeded;
			bBusy := FALSE;
			RETURN;
		END_IF
		nZFeedSum := nZFeedSum + nZFeed;
		IF nZFeedSum <= nZFeedMax THEN	//Feed auf begrenzen
			nZFeed := nZFeedSum - nZFeedMax;
			nZFeedSum := nZFeedMax;
			//letzter Move
			bMaxFeedAchieved := TRUE;
		END_IF

		MEMSET(ADR(stActionData),0,SIZEOF(stActionData));
		stActionData.eAction := E_Action.ACTION_MoveZ;
		stActionData.aParams[1] := E_MoveMode.MODE_Relative;
		stActionData.aParams[2] := nZFeed;	//Verfahrweg in Z
		stActionData.aParams[3] := -1;	//Speed		
		nErrorId := pMzTool^.M_ExeAction(stActionData);
		nState := 3;
		
	3:	//Warten bis ZMove fertig
		IF NOT pMzTool^.M_GetActionBusy(E_Action.ACTION_MoveZ) THEN
			nState := 1;
		END_IF
		
	4:	//XMove auf Mittelwert der beiden Probe-Werte
		MEMSET(ADR(stActionData),0,SIZEOF(stActionData));
		stActionData.eAction := E_Action.ACTION_MoveX;
		stActionData.aParams[1] := E_MoveMode.MODE_AbsNoneOffset;
		stActionData.aParams[2] := REAL_TO_DINT((rCapturedPos1 + rCapturedPos2) / 2);
		stActionData.aParams[3] := -1; //FastSpeed
		stActionData.aParams[4] := 1;	//Z-Kollision ignorieren
		nErrorId := pMzTool^.M_ExeAction(stActionData);
		nState := 5;
		
	5:	//Warten bis XMove fertig
		IF NOT pMzTool^.M_GetActionBusy(E_Action.ACTION_MoveX) THEN
			stProbePos := pMzTool^.P_stCurrentPosPhys;
			IF pTipCalibrator^.P_bXSensor THEN //steht nicht auf Sensor
				bBeginStartPos := TRUE;
				bSingleProbe := TRUE;
				nZFeed := 100;
				bProbeFlag := TRUE;
				nState := 7;	
			ELSE	//steht auf Sensor
				//in Z nach oben fahren
				MEMSET(ADR(stActionData),0,SIZEOF(stActionData));
				stActionData.eAction := E_Action.ACTION_MoveZ;
				stActionData.aParams[1] := E_MoveMode.MODE_Relative;
				stActionData.aParams[2] := 5000;	//Verfahrweg in Z
				stActionData.aParams[3] := 1600;	//Speed		
				nErrorId := pMzTool^.M_ExeAction(stActionData);
				nState := 6;
			END_IF
		END_IF
		
	6:	//Warten bis ZMove fertig oder Sensor
		IF pTipCalibrator^.P_bXSensor THEN	//Stoppen
			stActionData.eAction := E_Action.ACTION_Stop;
			nErrorId := pMzTool^.M_ExeAction(stActionData);
		END_IF
		
		IF NOT pMzTool^.M_GetActionBusy(E_Action.ACTION_MoveZ) THEN
			bBeginStartPos := TRUE;
			nZFeed := 100;
			bProbeFlag := TRUE;
			nState := 7;
		END_IF

	7:	//Probe ob oberhalb oder unterhalb Sensor	
		A_ProbeX();
		IF nStateA_ProbeX = 80 THEN
			nStateA_ProbeX := 0;
			bBeginStartPos := FALSE;
			IF bProbeFlag THEN	//wurde noch nicht nach unten getaktet
				bProbeFlag := FALSE;
				IF bProbeSuccess THEN	//steht unterhalb Sensor muss also nach oben
					nState := 8;
				ELSE //steht oberhalb Sensor
					nZFeed := -nZFeed;
					nState := 8;
				END_IF
			ELSE //es wurde bereits nach unten getaktet
				IF bProbeMissingTouch THEN //es wurde nach oben getaktet
					IF bProbeSuccess THEN
						//wieder nach unten takten, aber mit halber Schrittweite
						nZFeed := -nZFeed / 2;
					END_IF
				ELSE //es wurde nach unten getaktet
					IF bProbeSuccess THEN
						IF nZFeed >= nZFeedEnde THEN
							IF bProbePositiveOK AND bProbeNegativeOK THEN
								stTempPoint := pMzTool^.P_stCurrentPosPhys;
								stProbePos.Z := stTempPoint.Z;
								bBusy := FALSE;
							ELSE
								RETURN;
							END_IF
						END_IF
						nZFeed := -nZFeed / 2;
					END_IF
				END_IF
				nState := 8;
			END_IF
		ELSIF nStateA_ProbeX = 99 THEN
			nStateA_ProbeX := 0;
			bBusy := FALSE;
			bError := TRUE;
			nErrorId := nProbeErrorId;
		END_IF

	8:	//ZMove
		nZFeedSum := nZFeedSum + nZFeed;
		IF nZFeedSum < (nZFeedMax -100) THEN
			nErrorId := E_ErrorIdCmd.ERRORID_MeasureZDistanceExeeded;
			bError := TRUE;
			bBusy := FALSE;
			RETURN;
		END_IF	
		MEMSET(ADR(stActionData),0,SIZEOF(stActionData));
		stActionData.eAction := E_Action.ACTION_MoveZ;
		stActionData.aParams[1] := E_MoveMode.MODE_Relative;
		stActionData.aParams[2] := nZFeed;	//Verfahrweg in Z
		stActionData.aParams[3] := -1;	//Speed		
		nErrorId := pMzTool^.M_ExeAction(stActionData);
		nState := 9;
		
	9:	//Warten bis ZMove fertig
		IF NOT pMzTool^.M_GetActionBusy(E_Action.ACTION_MoveZ) THEN
			IF nZFeed < 0 THEN
				bProbeMissingTouch := FALSE;
 			ELSE
				bProbeMissingTouch := TRUE;
				bSingleProbe := TRUE;
			END_IF
			nState := 7;
		END_IF
		
	70:	//Abbrechen
		IF nStateA_ProbeX > 0 THEN
			nStateA_ProbeX := 70;
			A_ProbeX();
			nState := 71;
		ELSIF nStateA_ProbeY > 0 THEN
			nStateA_ProbeY := 70;
			A_ProbeY();
			nState := 72;
		ELSIF pMzTool^.M_GetActionBusy(E_Action.ACTION_MoveX) THEN
			pMzTool^.M_CancelAction(E_Action.ACTION_MoveX);
		ELSIF pMzTool^.M_GetActionBusy(E_Action.ACTION_MoveZ) THEN
			pMzTool^.M_CancelAction(E_Action.ACTION_MoveZ);
		ELSE
			bBusy := FALSE;
		END_IF
	
	71:	
		A_ProbeX();
		IF nStateA_ProbeX >= 80 THEN
			IF nStateA_ProbeX >= 99 THEN
				bError := TRUE;
			END_IF
			nStateA_ProbeX := 0;
			bBusy := FALSE;
		END_IF

	72:
		A_ProbeY();
		IF nStateA_ProbeY >= 80 THEN
			IF nStateA_ProbeY >= 99 THEN
				bError := TRUE;
			END_IF
			nStateA_ProbeY := 0;
			bBusy := FALSE;
		END_IF			
END_CASE
END_ACTION

ACTION A_ProbeX:
CASE nStateA_ProbeX OF
	0:		
		pXDrive := pMzTool^.P_pXDrive;
		IF pXDrive = 0 THEN
			nStateA_ProbeX := 99;
			RETURN;
		END_IF
		
		IF bBeginStartPos THEN	//MoveX zum Startpunkt
			MEMSET(ADR(stActionData),0,SIZEOF(stActionData));
			stActionData.eAction := E_Action.ACTION_MoveX;
			stActionData.aParams[1] := E_MoveMode.MODE_AbsWithOffset;
			stActionData.aParams[2] := nStartPos;
			stActionData.aParams[3] := -1; //FastSpeed
			stActionData.aParams[4] := 1;	//Z-Kollision ignorieren
			nProbeErrorId := pMzTool^.M_ExeAction(stActionData);
			bDirPositive := FALSE; //erste Richtung festlegen
			bProbePositiveOK := FALSE;
			bProbeNegativeOK := FALSE;
			MEMSET(ADR(stTempPoint),0,SIZEOF(stTempPoint));
			nStateA_ProbeX := 1;
		ELSE
			bDirPositive := NOT bDirPositive; //Richtung umkehren
			IF bDirPositive THEN
				bProbePositiveOK := FALSE;
			ELSE
				bProbeNegativeOK := FALSE;
			END_IF
			nStateA_ProbeX := 2;
		END_IF
			nProbeCount := 0;
			bProbeSuccess := FALSE;

	1:	//Warte	bis MoveX fertig
		IF NOT pMzTool^.M_GetActionBusy(E_Action.ACTION_MoveX) THEN
			nStateA_ProbeX := 2;
		END_IF

	2:	//XMove mit TouchProbe
		pXDrive^.M_Capture();
		bTouchProbe := FALSE;
		MEMSET(ADR(stActionData),0,SIZEOF(stActionData));
		stActionData.eAction := E_Action.ACTION_MoveX;
		stActionData.aParams[1] := E_MoveMode.MODE_AbsWithOffset;
		IF bDirPositive THEN	//XMove Richtung StartPos
			stActionData.aParams[2] := nStartPos;
		ELSE  //XMove Richtung EndPos
			stActionData.aParams[2] := nEndPos;
		END_IF
		stActionData.aParams[3] := nProbeSpeed;	//Speed
		stActionData.aParams[4] := 1;	//Z-Kollision ignorieren
		nProbeErrorId := pMzTool^.M_ExeAction(stActionData);		
		nStateA_ProbeX := 3;
		
	3:	//Warte	bis MoveX fertig
		IF NOT pMzTool^.M_GetActionBusy(E_Action.ACTION_MoveX) THEN
			//Sensor darf jetzt nicht geschalten sein
			IF NOT pTipCalibrator^.P_bXSensor THEN
				nProbeErrorId := E_ErrorIdCmd.ERRORID_TipCalibSensor;
				pXDrive^.M_StopCapture();
				nStateA_ProbeX := 99;
				RETURN;
			END_IF
			nProbeCount := nProbeCount  + 1;
			IF pXDrive^.P_bCaptureOk THEN
				bTouchProbe := TRUE;
			END_IF
			IF bProbeMissingTouch THEN	//es wird auf fehlendes Signal getesten
				bProbePositiveOK := FALSE;
				bProbeNegativeOK := FALSE;
				IF bTouchProbe THEN	 //nicht erfolgreich
					nStateA_ProbeX := 80;	//Fertig!!
				ELSE
					IF bSingleProbe THEN  //erfolgreich
						bProbeSuccess := TRUE;
						pXDrive^.M_StopCapture();
						nStateA_ProbeX := 10;	//Fertig!!//TouchProbe zurücksetzen
					ELSE
						IF nProbeCount = 1 THEN
							//Zweiter Move - TouchProbe nicht zurücksetzen
							bDirPositive := NOT bDirPositive; //Richtung umkehren
							nStateA_ProbeX := 2;  //XMove
						ELSE
							bProbeSuccess := TRUE;
							pXDrive^.M_StopCapture();
							nStateA_ProbeX := 10;	//Fertig!!//TouchProbe zurücksetzen
						END_IF
					END_IF
				END_IF
			ELSE	//es wird auf kommendes Signal getestet
				IF bTouchProbe THEN	//Signal ist gekommen
					IF bDirPositive THEN
						rCapturedPos1 := pXDrive^.P_rCapturedPos;
						stTempPoint.X := rCapturedPos1;
						stTempPoint := pMzTool^.M_RawPosToRealPos(stTempPoint);
						nEndPos := REAL_TO_DINT(stTempPoint.X - 1500);
						bProbePositiveOK := TRUE;
					ELSE
						rCapturedPos2 := pXDrive^.P_rCapturedPos;
						stTempPoint.X := rCapturedPos2;
						stTempPoint := pMzTool^.M_RawPosToRealPos(stTempPoint);
						nStartPos := REAL_TO_DINT(stTempPoint.X + 1500);
						bProbeNegativeOK := TRUE;
					END_IF
					
					IF bSingleProbe THEN //erfolgreich
						bProbeSuccess := TRUE;
						nStateA_ProbeX := 80;	//Fertig!!
					ELSE //TwinProbe
						IF nProbeCount = 1 THEN //war erster Move
							//Zweiter Move erforderlich
							bDirPositive := NOT bDirPositive; //Richtung umkehren
							nStateA_ProbeX := 2;  //XMove
						ELSE
							bProbeSuccess := TRUE;
							nStateA_ProbeX := 80;	//Fertig!!
						END_IF
					END_IF
				ELSE //Signal ist nicht gekommen
					IF bSingleProbe THEN //SingleProbe - nicht erfolgreich
						pXDrive^.M_StopCapture();
						nStateA_ProbeX := 10;	//Fertig!!//TouchProbe zurücksetzen
					ELSE //TwinProbe
						IF nProbeCount = 1 THEN //war erster Move
							//Zweiter Move
							bDirPositive := NOT bDirPositive; //Richtung umkehren
							nStateA_ProbeX := 2;  //XMove
						ELSE //war zweiter Move -> nicht erfolgreich
							pXDrive^.M_StopCapture();
							nStateA_ProbeX := 90;	//Fertig!!//TouchProbe zurücksetzen
						END_IF
					END_IF
				END_IF
			END_IF
		END_IF
		
	70:	//Abbrechen
		IF pMzTool^.M_GetActionBusy(E_Action.ACTION_MoveX) THEN
			pMzTool^.M_CancelAction(E_Action.ACTION_MoveX);
			pXDrive^.M_StopCapture();
		ELSE
			nStateA_ProbeX := 80;
		END_IF
		

	10,90:	//TouchProbe zurücksetzen
		IF pXDrive^.P_bCaptureStopped THEN
			IF nStateA_ProbeX = 10 THEN
				nStateA_ProbeX := 80;
			ELSE
				nStateA_ProbeX := 99;	
			END_IF
		END_IF
END_CASE

IF (nProbeErrorId > 0) AND (nStateA_ProbeX < 99) THEN
	pXDrive^.M_StopCapture();
	nStateA_ProbeX := 90;
END_IF
END_ACTION

ACTION A_ProbeY:
CASE nStateA_ProbeY OF
	0:	
		pYDrive := pMzTool^.P_pYDrive;
		IF pYDrive = 0 THEN
			nStateA_ProbeY := 99;
			RETURN;
		END_IF

		bDirPositive := TRUE;
		nProbeCount := 0;
		nStateA_ProbeY := 1;
		
	1:	//YMove	
		pYDrive^.M_Capture();
		bProbeSuccess := FALSE;
		bTouchProbe := FALSE;
		MEMSET(ADR(stActionData),0,SIZEOF(stActionData));
		stActionData.eAction := E_Action.ACTION_MoveY;
		stActionData.aParams[1] := E_MoveMode.MODE_AbsWithOffset;
		IF bDirPositive THEN	//XMove Richtung StartPos
			stActionData.aParams[2] := nEndPos;
		ELSE  //XMove Richtung EndPos
			stActionData.aParams[2] := nStartPos;
		END_IF
		stActionData.aParams[3] := nProbeSpeed;	//Speed
		stActionData.aParams[4] := 1;	//Z-Kollision ignorieren
		nProbeErrorId := pMzTool^.M_ExeAction(stActionData);	//ErrorHandling am Ende	
		nStateA_ProbeY := 2;
		
	2:	//Warte	bis MoveY fertig
		IF NOT pMzTool^.M_GetActionBusy(E_Action.ACTION_MoveY) THEN
			IF NOT pTipCalibrator^.P_bYSensor THEN
				nProbeErrorId := E_ErrorIdCmd.ERRORID_TipCalibSensor;
				pYDrive^.M_StopCapture();
				nStateA_ProbeY := 99;
				RETURN;
			END_IF
			
			nProbeCount := nProbeCount  + 1;
			IF pYDrive^.P_bCaptureOk THEN
				bTouchProbe := TRUE;
				pYDrive^.M_StopCapture();
			END_IF
							
			//es wird auf kommendes Signal getestet
			IF bTouchProbe THEN	//Signal ist gekommen
				IF bDirPositive THEN
					rCapturedPos1 := pYDrive^.P_rCapturedPos;
					bProbePositiveOK := TRUE;
				ELSE
					rCapturedPos2 := pYDrive^.P_rCapturedPos;;
					bProbeNegativeOK := TRUE;
				END_IF
				
				IF nProbeCount = 1 THEN //war erster Move
					//Zweiter Move erforderlich
					bDirPositive := NOT bDirPositive; //Richtung umkehren
					nStateA_ProbeY := 1;  //neuer YMove
				ELSE
					bProbeSuccess := TRUE;
					nStateA_ProbeY := 80;	//Fertig!!
				END_IF
			ELSE
				//Error (in Y muss in jedem Fall Probe positiv ausfallen)
				pYDrive^.M_StopCapture();
				nProbeErrorId := E_ErrorIdCmd.ERRORID_TipCalibProbeSensorY;
				nStateA_ProbeY := 90;
			END_IF
		END_IF
		
	70:	//Abbrechen
		IF pMzTool^.M_GetActionBusy(E_Action.ACTION_MoveY) THEN
			pMzTool^.M_CancelAction(E_Action.ACTION_MoveY);
			pYDrive^.M_StopCapture();
		ELSE
			nStateA_ProbeY := 80;
		END_IF
		

	10,90:	//TouchProbe zurücksetzen
		IF pYDrive^.P_bCaptureStopped THEN
			IF nStateA_ProbeY = 10 THEN
				nStateA_ProbeY := 80;
			ELSE
				nStateA_ProbeY := 99;	
			END_IF
		END_IF		
END_CASE

IF (nProbeErrorId > 0) AND (nStateA_ProbeY < 99) THEN
	pYDrive^.M_StopCapture();
	nStateA_ProbeY := 90;
END_IF
END_ACTION

METHOD M_Cancel
VAR_INPUT
END_VAR
IF bExecute AND nState < 70 THEN
	nState := 70;
END_IF
END_METHOD

END_FUNCTION_BLOCK

// ---- Actions/FB_MoveToTarget.TcPOU
FUNCTION_BLOCK FB_MoveToTarget
VAR_INPUT
	bExecute 	: BOOL;
	bStop		: BOOL;
END_VAR
VAR_OUTPUT
	bBusy		: BOOL;
	bError		: BOOL;
	nErrorId	: ERRORID;
END_VAR
VAR
	nState 		: USINT;
	pParamsChecked : BOOL;
	
	pMzTool				: POINTER TO FB_MzBase;
	pTwinPiezoHolder	: POINTER TO FB_TwinPiezoHolder;
	pTarget				: POINTER TO FB_TargetBase;
	pHighestTarget		: POINTER TO FB_TargetBase;
	pMtp				: POINTER TO FB_Mtp;
	pCustomUnitType1	: POINTER TO FB_CustomUnitType1;
	
	stPosition			: ST_3DPoint;
	stCurrentPosition	: ST_3DPoint;
	rectangle			: FB_Rectangle;
	bSuppressMoveFree	: BOOL;
	pCoHead				: POINTER TO FB_MzHead;
	
	eTargetRef				: E_TargetRef;
	nCol					: UINT;
	nRow					: UINT;
	nArrayNr				: USINT;
	nSpeedX					: DINT;
	nSpeedY					: DINT;
	nSpeedZ					: DINT;
	stOffset				: ST_3DPoint;
	nZLevel					: USINT;
	nIgnoreSlideAlignment	: USINT;
	stActionData			: ST_ActionData;
END_VAR

IF bExecute THEN
	IF nState = 0 THEN
		IF NOT pParamsChecked THEN
			nErrorId := 222;
			nState := 99;
		ELSE
			bBusy := TRUE;
			nState := 1;
		END_IF
	ELSE
		IF pMzTool^.P_bError THEN
			nErrorId := pMzTool^.P_nErrorId;
			nState := 99;
		END_IF
	END_IF
	
	//wenn TwinPiezoHolder, dann freifahren und einschwenken
	//wenn Pipette und deren Parent ein TwinPiezoHolder dann freifahren und ausschwenken
	IF nState = 1 THEN
		stCurrentPosition := pMzTool^.P_stCurrentPosTotal;
		bSuppressMoveFree := FALSE;
		IF pMzTool^.P_eObjectType = E_ObjectType.OBJECTTYPE_MZHead THEN
			nState := 6;	//gleich zum Freifahren
		ELSIF pMzTool^.P_eObjectType = E_ObjectType.OBJECTTYPE_TwinPiezoHolder THEN
			pTwinPiezoHolder := pMzTool;
			IF pTwinPiezoHolder^.P_eCurrentSwivelState = E_SwivelState.Swiveled THEN
				nState := 3;
			ELSE	//einschwenken			
				stActionData.eAction := E_Action.ACTION_Swivel;
				stActionData.aParams[1] := 1;
				nErrorId := pTwinPiezoHolder^.M_ExeAction(stActionData);
				IF nErrorId > 0 THEN
					nState := 99;
				ELSE
					nState := 2;
				END_IF
			END_IF
		ELSIF pMzTool^.P_eObjectType = E_ObjectType.OBJECTTYPE_PiezoPip AND pMzTool^.P_pParentMzTool^.P_eObjectType = E_ObjectType.OBJECTTYPE_TwinPiezoHolder THEN
			pTwinPiezoHolder := pMzTool^.P_pParentMzTool;
			IF pTwinPiezoHolder^.P_eCurrentSwivelState = E_SwivelState.Original THEN
				nState := 3;
			ELSE	//ausschwenken	
				stActionData.eAction := E_Action.ACTION_Swivel;
				stActionData.aParams[1] := 0;
				nErrorId := pTwinPiezoHolder^.M_ExeAction(stActionData);
				IF nErrorId > 0 THEN
					nState := 99;
				ELSE
					nState := 2;
				END_IF
			END_IF
		ELSE
			nState := 3;
		END_IF
	ELSIF nState = 2 THEN
		IF NOT pTwinPiezoHolder^.M_GetActionBusy(E_Action.ACTION_Swivel) THEN
			IF pTwinPiezoHolder^.P_bError THEN
				nErrorId := pTwinPiezoHolder^.P_nErrorId;
				nState := 99;
			ELSE
				nState := 3;
			END_IF
		END_IF
	END_IF
	
	//Falls ZielposZ höher als Freepos, dann vorher in Z auf Zielpos fahren
	//Das sollte auch geschehen, wenn Tool selber nicht freifahren muss.
	//Deshalb diese Überprüfung vorher erledigen
	IF nState = 3 THEN
		IF bStop THEN
			nState := 80;
		ELSE
			IF (pMzTool^.P_pMzHead^.P_bIsTopHead) AND
				(stPosition.Z > pTarget^.P_pWorkplate^.P_rCollHeight) AND
				stPosition.Z > stCurrentPosition.Z THEN
				nState := 4; //MoveZ
			ELSE
				nState := 6; //Entscheidung, wer Freifahrt übernimmt
			END_IF
		END_IF
	END_IF
	
	//Begin MoveZ
	IF nState = 4 THEN
		MEMSET(ADR(stActionData),0,SIZEOF(stActionData));
		stActionData.eAction := E_Action.ACTION_MoveZ;
		stActionData.aParams[1] := E_MoveMode.MODE_AbsWithOffset;
		stActionData.aParams[2] := REAL_TO_DINT(stPosition.Z);
		stActionData.aParams[3] := -1;
		nErrorId := pMzTool^.M_ExeAction(stActionData);
		IF nErrorId > 0 THEN
			nState := 99;
		ELSE
			nState := 5;
		END_IF
	ELSIF nState = 5 THEN
		IF bStop THEN
			pMzTool^.M_CancelAction(E_Action.ACTION_MoveZ);
			nState := 79;
		ELSE
			IF NOT pMzTool^.M_GetActionBusy(E_Action.ACTION_MoveZ) THEN
				nState := 6; //Entscheidung, wer Freifahrt übernimmt
			END_IF
		END_IF		
	END_IF
	//End MoveZ
	
	//Entscheidung, ob Freifahren hier oder durch MoveXY des Tools übernommen wird.
	IF nState = 6 THEN
		IF pTarget^.P_eObjectType = E_ObjectType.OBJECTTYPE_SpotArray THEN
			stCurrentPosition := pMzTool^.P_stCurrentPosTotal;
			//Überprüfen, ob Tool schon über diesem Target steht
			rectangle.M_Clear();
			rectangle.X1 := stCurrentPosition.X - 10;
			rectangle.X2 := stCurrentPosition.X + 10;
			rectangle.Y1 := stCurrentPosition.Y - 10;
			rectangle.Y2 := stCurrentPosition.Y + 10;
			IF F_RectIntersectRect(rectangle,pTarget^.P_fbAbsRect) THEN
				bSuppressMoveFree := TRUE;
				nState := 7;
			ELSE
				nState := 9;
			END_IF
		ELSE
			nState := 9;
		END_IF			
	END_IF
	
	//Begin MoveFree
	IF nState = 7 THEN
		nState := 9;
		IF NOT pMzTool^.P_pMzHead^.P_bCollFree THEN
			nState := 8;
			pMzTool^.P_pMzHead^.M_MoveFree(pMzTool);
		END_IF
		pCoHead := pMzTool^.P_pMzHead^.P_pCoHead;
		IF pCoHead > 0 AND_THEN NOT pCoHead^.P_bCollFree THEN
			nState := 8;
			pCoHead^.M_MoveFree(0);
		END_IF		
	ELSIF nState = 8 THEN
		nState := 9;
		IF pMzTool^.P_pMzHead^.M_GetActionBusy(E_Action.ACTION_MoveZ) THEN
			nState := 8;
		END_IF
		IF pCoHead > 0 AND_THEN pCoHead^.M_GetActionBusy(E_Action.ACTION_MoveZ) THEN
			nState := 8;
		END_IF
	END_IF
	//End MoveFree
	
	//Begin MoveXY
	IF nState = 9 THEN
		IF bStop THEN
			nState := 80;
		ELSE
			nState := 10;
			stActionData.eAction := E_Action.ACTION_MoveXY;
			stActionData.aParams[1] := E_MoveMode.MODE_AbsWithOffset;
			stActionData.aParams[2] := REAL_TO_DINT(stPosition.X);
			stActionData.aParams[3] := REAL_TO_DINT(stPosition.Y);
			stActionData.aParams[4] := nSpeedX;
			stActionData.aParams[5] := nSpeedY;
			stActionData.aParams[7] := 0; //nicht synchron
			IF bSuppressMoveFree THEN
				stActionData.aParams[6] := E_CrashAvoidanceMode.MoveNoneFree;
			ELSE
				stActionData.aParams[6] := E_CrashAvoidanceMode.MoveAllFree;
			END_IF
			
			nErrorId := pMzTool^.M_ExeAction(stActionData);
			IF nErrorId > 0 THEN
				nState := 99;
			END_IF			
		END_IF		
	ELSIF nState = 10 THEN
		IF bStop THEN
			pMzTool^.M_CancelAction(E_Action.ACTION_MoveXY);
			nState := 79;
		ELSE
			IF NOT pMzTool^.M_GetActionBusy(E_Action.ACTION_MoveXY) THEN
				IF pMzTool^.P_eObjectType = E_ObjectType.OBJECTTYPE_MZHead  OR pMzTool^.P_bCanceled THEN
					nState := 80;
				ELSE	//MoveZ
					nState := 11;
				END_IF
			END_IF
		END_IF		
	END_IF
	//End MoveXY
	
	//Begin MoveZ
	IF nState = 11 THEN
		IF nSpeedZ > 0 OR nSpeedZ = -1 THEN
			MEMSET(ADR(stActionData),0,SIZEOF(stActionData));
			stActionData.eAction := E_Action.ACTION_MoveZ;
			stActionData.aParams[1] := E_MoveMode.MODE_AbsWithOffset;
			stActionData.aParams[2] := REAL_TO_DINT(stPosition.Z);
			stActionData.aParams[3] := nSpeedZ;
			stActionData.aParams[4] := 5; //CollFreeAreaXMinus
			stActionData.aParams[5] := 5; //CollFreeAreaXPlus
			stActionData.aParams[6] := 5; //CollFreeAreaYMinus
			stActionData.aParams[7] := 5; //CollFreeAreaYPlus
			nErrorId := pMzTool^.M_ExeAction(stActionData);
			IF nErrorId > 0 THEN
				nState := 99;
			ELSE
				nState := 12;
			END_IF
		ELSE
			nState := 80;
		END_IF		
	ELSIF nState = 12 THEN
		IF bStop THEN
			pMzTool^.M_CancelAction(E_Action.ACTION_MoveZ);
			nState := 79;
		ELSE
			IF NOT pMzTool^.M_GetActionBusy(E_Action.ACTION_MoveZ) THEN
				nState := 80;
			END_IF			
		END_IF		
	END_IF
	//End MoveZ
	
	IF nState = 79 THEN
		IF NOT (pMzTool^.M_GetActionBusy(E_Action.ACTION_MoveZ) OR pMzTool^.M_GetActionBusy(E_Action.ACTION_MoveXY)) THEN
			nState := 80;
		END_IF
	END_IF
	
		
	IF nState >= 80 THEN
		bBusy := FALSE;
		IF nState = 99 THEN
			bError := TRUE;	
		END_IF
	END_IF
	
ELSE
	pParamsChecked := FALSE;
	nState := 0;
	bError := FALSE;
	bStop := FALSE;
	bBusy := FALSE;
END_IF

METHOD M_SetAndCheckParams : ERRORID
VAR_INPUT
	refActionData : REFERENCE TO ST_ActionData;
END_VAR

VAR
	i : UINT;
	//stPieceDimension : ST_3DDimension;
	rect : FB_Rectangle;
	//rToolRadius : REAL;
	stAbsPos : ST_3DPoint;
	bRiskOfCrash : BOOL;
END_VAR
IF bBusy THEN
	M_SetAndCheckParams := E_ErrorIdCmd.ERRORID_ComplexActionActive;  //Error
	RETURN;
END_IF

eTargetRef := DINT_TO_USINT(refActionData.aParams[1]);
nCol := DINT_TO_UINT(refActionData.aParams[2]);
nRow := DINT_TO_UINT(refActionData.aParams[3]);
nArrayNr := DINT_TO_USINT(refActionData.aParams[4]);
nSpeedX := refActionData.aParams[5];
nSpeedY := refActionData.aParams[6];
nSpeedZ := refActionData.aParams[7];
stOffset.X := DINT_TO_REAL(refActionData.aParams[8]);
stOffset.Y := DINT_TO_REAL(refActionData.aParams[9]);
stOffset.Z := DINT_TO_REAL(refActionData.aParams[10]);
nZLevel := DINT_TO_USINT(refActionData.aParams[11]);
nIgnoreSlideAlignment := DINT_TO_USINT(refActionData.aParams[12]);

IF NOT fbObjectDirectory.M_ObjIsMzTool(refActionData.nObject) THEN //Object gültiges MzTool?
	M_SetAndCheckParams := E_ErrorIdCmd.ERRORID_UnsuitableObject;  //Error
	RETURN;
END_IF
pMzTool := fbObjectDirectory.M_GetObjPointer(refActionData.nObject);

IF NOT fbObjectDirectory.M_ObjIsTarget(refActionData.nTarget) THEN //Gültiges Target?
	M_SetAndCheckParams := E_ErrorIdCmd.ERRORID_UnsuitableTarget;  //Error
	RETURN;
END_IF
pTarget := fbObjectDirectory.M_GetObjPointer(refActionData.nTarget);

//MzTool bereit für MoveToTarget?
M_SetAndCheckParams := pMzTool^.M_CheckAction(refActionData,0); 
IF  M_SetAndCheckParams > 0 THEN
	RETURN;
END_IF

//Target bereit für Action?
M_SetAndCheckParams := pTarget^.M_CheckAction(refActionData,0);
IF  M_SetAndCheckParams > 0 THEN
	RETURN;
END_IF

//absolute Position aus Target holen
stPosition := pTarget^.M_GetAbsPos(pChildPos:= 0, eTargetRef:= eTargetRef, 
									nParam1:= nCol,
									nParam2:= nRow,
									nParam3:= nArrayNr,
									nParam4:= nIgnoreSlideAlignment,
									nZLevel:= nZLevel, nErrorId=> nErrorId);									
									
IF nErrorId > 0 THEN
	M_SetAndCheckParams := nErrorId;
	RETURN;
END_IF
//Offset addieren
stPosition := F_Add3DPoints(stPosition, stOffset);

//Check Speed
//Falls SpeedX oder SpeedY "0" sind dann Z auch auf "0" setzen
IF nSpeedX = 0 OR nSpeedY = 0 THEN
	nSpeedZ := 0;
END_IF	

//Position auf Limits checken
//Targetposition X auf Limits checken
IF nSpeedX <> 0 THEN
	IF NOT pMzTool^.M_CheckMoveLimit(sAxis:= 'X', eMoveMode:= E_MoveMode.MODE_AbsWithOffset,rMovePosition:= stPosition.X) THEN
		M_SetAndCheckParams := E_ErrorIdCmd.ERRORID_TargetPosOutOfRangeX;
		RETURN;
	END_IF
END_IF
//Targetposition Y auf Limits checken
IF nSpeedY <> 0 THEN
	IF NOT pMzTool^.M_CheckMoveLimit(sAxis:= 'Y', eMoveMode:= E_MoveMode.MODE_AbsWithOffset,rMovePosition:= stPosition.Y) THEN
		M_SetAndCheckParams := E_ErrorIdCmd.ERRORID_TargetPosOutOfRangeY;
		RETURN;
	END_IF
END_IF
//Targetposition Z auf Limits checken
IF nSpeedZ <> 0 THEN
	IF NOT pMzTool^.M_CheckMoveLimit(sAxis:= 'Z', eMoveMode:= E_MoveMode.MODE_AbsWithOffset,rMovePosition:= stPosition.Z) THEN
		M_SetAndCheckParams := E_ErrorIdCmd.ERRORID_TargetPosOutOfRangeZ;
		RETURN;
	END_IF
	//Das hier ist ein Provisorium!!
	IF pMzTool^.P_pMzHead^.P_bIsTopHead THEN
		FOR i:= 1 TO cMaxCustomUnitTyp1 BY 1 DO
			IF afbCustomUnitType1[i].P_nObjectID > 0 THEN
				stAbsPos := afbCustomUnitType1[i].P_stAbsPosCenter;
				IF stPosition.Z < stAbsPos.Z THEN
					(*IF pMzTool^.P_pPiece > 0 THEN
						stPieceDimension := pMzTool^.P_pPiece^.P_stDimension;
						rToolRadius := stPieceDimension.Width / 2.0;
					ELSE
						rToolRadius := 2000.0;
					END_IF*)
					rect.X1 := stPosition.X - pMzTool^.P_rToolRadius;
					rect.X2 := stPosition.X + pMzTool^.P_rToolRadius;
					rect.Y1 := stPosition.Y - pMzTool^.P_rToolRadius;
					rect.Y2 := stPosition.Y + pMzTool^.P_rToolRadius;
					//Zuerst checken, ob das Target selber in dem Bereich
					IF F_RectIntersectRect(rect,afbCustomUnitType1[i].P_fbAbsRect) THEN
						bRiskOfCrash := TRUE;
						IF afbCustomUnitType1[i].M_GetRectIsInnerSlot(rect) THEN
							bRiskOfCrash := FALSE;
							EXIT;
						END_IF
					END_IF
				END_IF
			END_IF
		END_FOR
	END_IF
	IF bRiskOfCrash THEN
		M_SetAndCheckParams := E_ErrorIdCmd.ERRORID_MoveZRiskOfCrash;
		RETURN;
	END_IF
END_IF
pParamsChecked := TRUE;
END_METHOD

END_FUNCTION_BLOCK

// ---- Objects/F_RectIntersectRect.TcPOU
FUNCTION F_RectIntersectRect : BOOL
VAR_INPUT
	stRect1 : FB_Rectangle;
	stRect2 : FB_Rectangle;
END_VAR
VAR
END_VAR

//schneidet Rechteck1 Rechteck2?
F_RectIntersectRect := TRUE;
IF stRect1.X1 > stRect2.X2 OR stRect2.X1 > stRect1.X2 THEN
	F_RectIntersectRect := FALSE;
END_IF

IF stRect1.Y1 > stRect2.Y2 OR stRect2.Y1 > stRect1.Y2 THEN
	F_RectIntersectRect := FALSE;
END_IF

END_FUNCTION

// ---- Error/FB_ErrorList.TcPOU
FUNCTION_BLOCK FB_ErrorList
VAR_INPUT
	putPosPtr	: POINTER TO T_LinkedListEntry := 0;(* Linked list node position pointer (used by A_Find, A_GetNext, A_GetPrev) *)
	putValue 	: ST_Error;(* Linked list nod value (used by A_AddHead, A_AddTail, A_Find )*)
END_VAR
VAR_OUTPUT
	bOk			: BOOL := FALSE;(* TRUE = Success, FALSE = Failed *)
	getPosPtr	: POINTER TO T_LinkedListEntry := 0;(* Returned linked list node position pointer *)
	getValue 	: ST_Error;(* Returned linked list node value *)
	nCount		: UDINT := 0;(* Linked list size (number of used nodes, used by A_Count) *)	
END_VAR
VAR
	dataPool		: ARRAY[0..10] OF ST_Error;(* Structured data element pool *)
	nodes			: ARRAY[0..10] OF T_LinkedListEntry;(* Max. number of linked list nodes. The value of list node = 32 bit integer (pointer to dataPool-array-entry) *)
	fbList 			: FB_LinkedListCtrl;(* basic linked list control function block *)
	hList 			: T_HLINKEDLIST;(* linked list handle *)
	pRefPtr			: POINTER TO ST_Error := 0;
	indexOfElem		: PVOID;
	nSumCount		: UINT;
END_VAR

ACTION A_Add:
putValue.MachineMode := MainDispacher.eCurrentMode;
putValue.MachineState := MainDispacher.P_eCurrentState;
putValue.TimeStamp := timeStamp;
(* Adds head to the node list *)
MEMSET( ADR( getValue ), 0, SIZEOF( getValue ) );
getPosPtr := 0;

fbList.A_AddHeadValue( hList := hList, putValue := 16#00000000(* we will set this value later *), getPosPtr=>getPosPtr, bOk=>bOk );(* Add new element to the list, getPosPtr points to the new list node *)
IF fbList.bOk THEN(* Success *)
	fbList.A_GetIndexAtPosPtr( hList := hList, putPosPtr := getPosPtr, getValue =>indexOfElem, bOk=>bOk );(* Get array index of getPosPtr *)
	IF fbList.bOk THEN(* Success *)
		pRefPtr 	:= ADR( dataPool[indexOfElem] );(* Get pointer to the data element *)
		pRefPtr^ := putValue;(* set element value *)

		fbList.A_SetValueAtPosPtr( hList := hList, putPosPtr := getPosPtr, putValue := pRefPtr, bOk=>bOk );(* Assign the node value = pointer to the data element *)
		IF fbList.bOk THEN(* Success *)
			getValue := putValue;
		END_IF
	END_IF
END_IF

nCount := hList.nCount;
END_ACTION

ACTION A_Get:
(* Gets tail node position pointer and value *)
MEMSET( ADR( getValue ), 0, SIZEOF( getValue ) );
getPosPtr := 0;

fbList.A_GetTail( hList := hList, getValue=>pRefPtr, getPosPtr=>getPosPtr, bOk=>bOk );
IF fbList.bOk THEN
	getValue := pRefPtr^;
END_IF
END_ACTION

ACTION A_Remove:
(* Remove tail node from node list *)
MEMSET( ADR( getValue ), 0, SIZEOF( getValue ) );
getPosPtr := 0;

fbList.A_RemoveTailValue( hList := hList, getValue=>pRefPtr, getPosPtr=>getPosPtr, bOk=>bOk );
IF fbList.bOk THEN
	getValue := pRefPtr^;
END_IF

nCount := hList.nCount;
END_ACTION

ACTION A_Reset:
(* Reset/initialize linked list *)
MEMSET( ADR( getValue ), 0, SIZEOF( getValue ) );
getPosPtr := 0;
bOk := F_CreateLinkedListHnd( ADR( nodes ), SIZEOF( nodes ), hList );(* Intialize list handle *)
fbList.A_Reset( hList := hList, bOk=>bOk );
nCount := 0;
END_ACTION

METHOD M_Add
VAR_INPUT
	stError	: ST_Error;
END_VAR
A_Add(putValue := stError);
END_METHOD

METHOD M_AddExt
VAR_INPUT
	nErrorId	: ERRORID;
	nErrorId2	: UDINT;
	HardwareGrp	: HARDWAREGRP;		//Hardwaregruppe, bei der der Fehler aufgetaucht ist
	HardwareNr	: UINT;				//Hardwarenummer, bei der der Fehler aufgetaucht ist
	POU			: E_POU;			//Baustein, in dem der Fehler aufgetreten ist
	POUAction	: E_POUACT;			//Methode bzw. Action, in der der Fehler aufgetreten ist
	POUState	: UINT;				//State der Statemachine, in der der Fehler aufgetreten ist
END_VAR
VAR
	stError : ST_Error;
END_VAR
stError.ErrorId := nErrorId;
stError.ErrorId2 := nErrorId2;
stError.HardwareGrp := HardwareGrp;
stError.HardwareNr := HardwareNr;
stError.POU := POU;
stError.POUAction := POUAction;
stError.POUState := POUState;
A_Add(putValue := stError);
END_METHOD

END_FUNCTION_BLOCK

// ---- Sequence/FB_SequenceList.TcPOU
FUNCTION_BLOCK FB_SequenceList
VAR_INPUT
END_VAR
VAR_OUTPUT
END_VAR
VAR
	pHead				: POINTER TO ST_Pointer;
	pTail				: POINTER TO ST_Pointer;
	pMonitorSequence 	: POINTER TO FB_Sequence;
	nCount				: UINT;
END_VAR

METHOD FB_exit : BOOL
VAR_INPUT
	bInCopyCode : BOOL; // if TRUE, the exit method is called for exiting an instance that is copied afterwards (online change).
END_VAR

VAR
	bFlag : BOOL;
END_VAR
REPEAT
	bFlag := M_Delete(); 
UNTIL  bFlag
END_REPEAT
END_METHOD

METHOD M_Add : BOOL
VAR_INPUT
	nId			: UDINT;
	nNoOfSteps	: UINT;
END_VAR

VAR
	nNoOfSteps1 : UINT;
	pNew 		: POINTER TO ST_Pointer;
	pTemp		: POINTER TO ST_Pointer;
	pSequence	: POINTER TO FB_Sequence;
END_VAR
//Überprüfen, ob Id schon vorhanden, wenn ja, dann löschen
pNew := pHead;
WHILE pNew > 0 DO
	pSequence := pNew^.pContent;
	IF pSequence^.P_nId = nId THEN	//Sequence schon vorhanden -> erst löschen
		IF pSequence^.M_Delete(nMaxSteps:= 200) THEN
			//Folgende Fälle können auftreten
			//1. es existiert nur eine Sequenz (pHead = pTail
			//->pHead und pTail auf "0"
			//2. pNew ist pHead
			//->pNext von pHead wird zu pHead, pHead.Prev wird 0
			//3. pNew ist 
			IF pNew = pHead THEN
				IF pNew^.pNext > 0 THEN
					pHead := pNew^.pNext;
					pHead^.pPrev := 0;
				ELSE
					pHead := 0;
					pTail := 0;
				END_IF
			ELSIF pNew = pTail THEN
				pTail := pTail^.pPrev;
				pTail^.pNext := 0;
			ELSE
				pTemp := pNew^.pPrev;
				pTemp^.pNext := pNew^.pNext;
				pTemp := pNew^.pNext;
				pTemp^.pPrev := pNew^.pPrev;
			END_IF
			__DELETE(pSequence);
			__DELETE(pNew);
			nCount := nCount - 1;
			EXIT;
		ELSE
			RETURN;
		END_IF
	ELSE
		pNew := pNew^.pNext;	
	END_IF
END_WHILE
nNoOfSteps1 := nNoOfSteps;
pSequence := __NEW(FB_Sequence(nNoOfSteps:= nNoOfSteps1));
pSequence^.P_nId := nId;
pNew := __NEW(ST_Pointer);
pNew^.pContent := pSequence;
IF pHead = 0 THEN
	pHead := pTail := pNew;
ELSE
	pNew^.pPrev := pTail; 
	pTail^.pNext := pNew;
	pTail := pNew;
END_IF
nCount := nCount + 1;
M_Add := TRUE;
END_METHOD

METHOD M_Delete : BOOL
VAR_INPUT
END_VAR
VAR
	pPointer  		: POINTER TO ST_POINTER;
	pSequence 		: POINTER TO FB_Sequence;
	nDelSteps 		: UINT;
	nDeletedSteps	: UINT;
END_VAR

VAR_INST
	
END_VAR

VAR CONSTANT
	cMaxSteps : UINT := 100;
END_VAR
//Alle Sequencen löschen
//Es sollen max. Steps pro Zyklus gelöscht werden
//M_Delete() gibt die Anzahl der gelöschten Steps zurück
pPointer := pHead;
WHILE pPointer > 0 DO
	pSequence := pPointer^.pContent;
	IF pSequence^.M_Delete(nMaxSteps:= (cMaxSteps - nDeletedSteps), nDeletedSteps=>nDelSteps) THEN	//Alle Step aus Sequence entfernt
		//aus Liste löschen
		//Der nächste wird zum Head
		IF pHead <> pTail THEN
			pHead := pHead^.pNext;
		ELSE
			pHead := pTail := 0;
		END_IF
		__DELETE(pSequence);
		__DELETE(pPointer);
	END_IF
	nDeletedSteps := nDeletedSteps + nDelSteps;
	IF (nDeletedSteps = cMaxSteps) AND (pHead > 0) THEN
		RETURN;
	END_IF
	pPointer := pHead;
END_WHILE
nDeletedSteps := 0;
nCount := 0;
M_Delete := TRUE;
END_METHOD

METHOD M_Get : POINTER TO FB_Sequence
VAR_INPUT
	nId : UDINT;
END_VAR

VAR
	pPointer	: POINTER TO ST_POINTER;
	pSequence	: POINTER TO FB_Sequence;
END_VAR
pPointer := pHead;
WHILE pPointer > 0 DO
	pSequence := pPointer^.pContent;
	IF pSequence^.P_nId = nId THEN
		M_Get := pSequence;
		RETURN;
	END_IF
	pPointer := pPointer^.pNext;
END_WHILE
END_METHOD

METHOD M_ResetAllSequ
VAR_INPUT
END_VAR
VAR
	pPointer  		: POINTER TO ST_POINTER;
	pSequence 		: POINTER TO FB_Sequence;
END_VAR
pPointer := pHead;
WHILE pPointer > 0 DO
	pSequence := pPointer^.pContent;
	pSequence^.M_Reset();
	pPointer := pPointer^.pNext;
END_WHILE
END_METHOD

END_FUNCTION_BLOCK

// ---- Sequence/FB_SequenceInfo.TcPOU
FUNCTION_BLOCK FB_SequenceInfo
VAR_INPUT
END_VAR
VAR_OUTPUT
END_VAR
VAR
	pHead : POINTER TO ST_Pointer;
	pTail : POINTER TO ST_Pointer;
END_VAR

METHOD M_AddTail
VAR_INPUT
	nSequenceNr		: UDINT;
	eSequenceState	: E_SequenceState;
	pStep			: POINTER TO ST_Step;
END_VAR

VAR
	pSeekPointer: POINTER TO ST_Pointer;
	pSeekContent: POINTER TO ST_SequenceInfo;		

	pNewPointer : POINTER TO ST_Pointer;
	pNewContent : POINTER TO ST_SequenceInfo;
END_VAR
IF pStep > 0 THEN
	IF pStep^.bInfoChanged THEN
		pSeekPointer := pHead; //Step schon mit geleichem State schon vorhanden? Wenn ja, dann nur Info überschreiben.
								//Bei Timern trat das Problem auf, dass mehr Infos generiert werden, als dass in dieser Zeit diese
								//auch ausgelesen werden.
		WHILE(pSeekPointer > 0) DO
			pSeekContent := pSeekPointer^.pContent;
			IF pSeekContent^.nStepNr = pStep^.nStepNr AND_THEN pSeekContent^.nSequId = nSequenceNr THEN
				IF pSeekContent^.eStepState = pStep^.eState AND pSeekContent^.eSequenceState = eSequenceState THEN
					//nur Info ändern
					pSeekContent^.nInfo := pStep^.nInfo;
					RETURN;
				END_IF
			END_IF
			pSeekPointer := pSeekPointer^.pNext;
		END_WHILE
		
		pNewPointer := __NEW(ST_Pointer);
		pNewContent := __NEW(ST_SequenceInfo);
		MEMSET(pNewPointer,0,SIZEOF(ST_Pointer));
		pNewContent^.nSequId := nSequenceNr;
		pNewContent^.eSequenceState := eSequenceState;
		pNewContent^.nStepNr := pStep^.nStepNr;
		pNewContent^.eStepState := pStep^.eState;
		pNewContent^.nInfo := pStep^.nInfo;
		pStep^.bInfoChanged := FALSE;
	ELSE
		RETURN;
	END_IF
ELSE
	pNewPointer := __NEW(ST_Pointer);
	pNewContent := __NEW(ST_SequenceInfo);
	MEMSET(pNewPointer,0,SIZEOF(ST_Pointer));
	pNewContent^.nSequId := nSequenceNr;
	pNewContent^.eSequenceState := eSequenceState;
	pNewContent^.nStepNr := 0;
	pNewContent^.eStepState := E_StepState.STEPSTATUS_Idle;
END_IF

pNewPointer^.pContent := pNewContent;

IF pTail = 0 THEN
	pHead := pTail := pNewPointer;
ELSE
	pNewPointer^.pPrev := pTail;
	pTail^.pNext := pNewPointer;
	pTail := pNewPointer;
END_IF
END_METHOD

METHOD M_GetHead
VAR_INPUT
END_VAR
VAR_IN_OUT
	stSequenceStatus : ST_SequenceInfo;
END_VAR

VAR
	pContent	: POINTER TO ST_SequenceInfo;
	pTemp		: POINTER TO ST_Pointer;
END_VAR
//Immer vom Head holen und dann löschen
IF pHead > 0 THEN
	MEMCPY(ADR(stSequenceStatus),pHead^.pContent,SIZEOF(ST_SequenceInfo));
	__DELETE(pHead^.pContent);
	IF pHead^.pNext > 0 THEN //Next wird zu Head
		pTemp := pHead^.pNext;
		__DELETE(pHead);
		pTemp^.pPrev := 0;
		pHead := pTemp;
	ELSE
		__DELETE(pHead);
		pTail := 0;
	END_IF
END_IF
END_METHOD

END_FUNCTION_BLOCK

// ---- Functions/F_CuboidInnerCuboid.TcPOU
FUNCTION F_CuboidInnerCuboid : BOOL
VAR_INPUT
	stCuboid1 : ST_Cuboid;
	stCuboid2 : ST_Cuboid;
END_VAR
VAR
END_VAR

F_CuboidInnerCuboid := (stCuboid1.stPos.X + stCuboid1.stDim.Width) > stCuboid2.stPos.X AND
						stCuboid1.stPos.X < (stCuboid2.stPos.X + stCuboid2.stDim.Width) AND
						(stCuboid1.stPos.Y + stCuboid1.stDim.Depth) > stCuboid2.stPos.Y AND
						stCuboid1.stPos.Y < (stCuboid2.stPos.Y + stCuboid2.stDim.Depth) AND  
						(stCuboid1.stPos.Z + stCuboid1.stDim.Height) > stCuboid2.stPos.Z AND
						stCuboid1.stPos.Y < (stCuboid2.stPos.Z + stCuboid2.stDim.Height);

END_FUNCTION

// ---- Functions/F_GET_GCODE_NCLINE.TcPOU
FUNCTION F_GET_GCODE_NCLINE : REAL
VAR_INPUT
	sGCodeLines: STRING(100);
	sSeachCode: STRING;
END_VAR
VAR
	nLines: USINT;
	nLenString: INT;
	nFirstPos: INT := 1;
	nEndPos: INT;
	i: INT;
	sLine: STRING(100);
	sChar: STRING(1);
	sValue: STRING;
END_VAR

nLenString := LEN(sGCodeLines);
//Anzahl der Zeilen ermitteln
REPEAT
	i := i + 1;
	IF MID(sGCodeLines,1,i) = '$N' THEN
		nLines := nLines + 1;
		IF nLines = 1 THEN
			nFirstPos := 1;
			nEndPos := i - 2;	
		ELSE
			nFirstPos := nEndPos + 3;
			nEndPos := i - 2;
		END_IF
	END_IF
UNTIL i = nLenString OR nLines = 3
END_REPEAT

IF nLines > 0 THEN
	sLine := MID(sGCodeLines, nEndPos - nFirstPos + 1, nFirstPos);
	//Nach Code suchen
	nFirstPos := FIND(sLine,sSeachCode);
	IF nFirstPos > 0 THEN
		IF sSeachCode = '@714' OR sSeachCode = '@717' THEN
				F_GET_GCODE_NCLINE := 1.0;
				RETURN;
		ELSIF sSeachCode = 'F' THEN
			i := nFirstPos;
			nLenString := LEN(sLine);
			//numerischen Wert nach F ermitteln
			REPEAT
				i := i + 1;
				sChar := MID(sLine,1,i);
				IF NOT ((sChar[0] > 47 AND sChar[0] < 58) OR sChar[0] = 46) OR i = nLenString THEN
					EXIT;
				ELSE
					sValue := CONCAT(sValue,sChar);
				END_IF
			UNTIL FALSE
			END_REPEAT
		END_IF		
	END_IF
END_IF
F_GET_GCODE_NCLINE := STRING_TO_REAL(sValue);

END_FUNCTION

// ---- Hardware/SimutateHwModules.TcPOU
PROGRAM SimutateHwModules
VAR
	stHardwareId : ST_HardwareId;
END_VAR

fbXDriveBeck.P_pMultiZRef := ADR(aFbMultiZRef[1]);
fbYDriveBeck.P_pMultiZRef := ADR(aFbMultiZRef[1]);
stHardwareId.eGroup := E_HardwareGrp.AxisX;
stHardwareId.nParentItem := 0;
stHardwareId.nItem := 1;
fbXDriveBeck.P_stHardwareId := stHardwareId;
stHardwareId.eGroup := E_HardwareGrp.AxisY;
stHardwareId.nParentItem := 1;
stHardwareId.nItem := 1;
fbYDriveBeck.P_stHardwareId := stHardwareId;
 
fbXYDriveList.M_Add(ADR(fbXDriveBeck));
fbXYDriveList.M_Add(ADR(fbYDriveBeck));

END_PROGRAM

// ---- Hardware/Trigger/OutDistributor.TcPOU
PROGRAM OutDistributor
VAR
	bInput1 AT%I* : BOOL;
	bInput2 AT%I* : BOOL;
	bInput3 AT%I* : BOOL;
	bInput4 AT%I* : BOOL;
	bOutput AT%Q* : BOOL;
END_VAR

bOutput := bInput1 OR bInput2 OR bInput3 OR bInput4;

END_PROGRAM

// ---- Objects/F_GetTwoLineAngle.TcPOU
FUNCTION F_GetTwoLineAngle : LREAL	//ermittelt den Winkel zwischen zwei Linien in XY-Ebene
VAR_INPUT
	line1_P1 : ST_3DPoint;
	line1_P2 : ST_3DPoint;
	line2_P1 : ST_3DPoint;
	line2_P2 : ST_3DPoint;	
END_VAR
VAR
	vec1X, vec1Y, vec2X, vec2Y : LREAL;
	temp : LREAL;
	angle1 : LREAL;
	angle2 : LREAL;
END_VAR

//1. Linien in Ortsvektoren umrechnen
vec1X := line1_P2.X - line1_P1.X;
vec1Y := line1_P2.Y - line1_P1.Y;

vec2X := line2_P2.X - line2_P1.X;
vec2Y := line2_P2.Y - line2_P1.Y;

//Vektor 1 auf Einheitskreis normalisieren
//Länge berechnen
temp := vec1X * vec1X + vec1Y * vec1Y;
IF temp = 0.0 THEN
	F_GetTwoLineAngle := 9999.9; //führt zu Wurzel aus "0" was bedeutet, dass der Vektor keine Länge hat
	RETURN;
END_IF
temp := SQRT(temp);
//normalisieren 
vec1X := vec1X / temp;
vec1Y := vec1Y / temp;

//Vektor 2 auf Einheitskreis normalisieren
//Länge berechnen
temp := vec2X * vec2X + vec2Y * vec2Y;
IF temp = 0.0 THEN
	F_GetTwoLineAngle := 9999.9; //führt zu Wurzel aus "0" was bedeutet, dass der Vektor keine Länge hat
	RETURN;
END_IF
temp := SQRT(temp);
//normalisieren 
vec2X := vec2X / temp;
vec2Y := vec2Y / temp;

//Winkelberechnung Vektor 1 in Bezug zu X-Achse im Koordinatensystem
IF vec1Y < 0.0 THEN	//Vektor befindet sich im Quadranten III oder IV
	angle1 := 360.0 -  RAD_TO_DEG(ACOS(vec1X));
ELSE
	angle1 := RAD_TO_DEG(ACOS(vec1X));
END_IF

//Winkelberechnung Vektor 2 in Bezug zu X-Achse im Koordinatensystem
IF vec2Y < 0.0 THEN	//Vektor befindet sich im Quadranten III oder IV
	angle2 := 360.0 -  RAD_TO_DEG(ACOS(vec2X));
ELSE
	angle2 := RAD_TO_DEG(ACOS(vec2X));
END_IF

F_GetTwoLineAngle := angle2 - angle1;

IF F_GetTwoLineAngle > 180.0 THEN
	F_GetTwoLineAngle := F_GetTwoLineAngle - 360.0;
END_IF

END_FUNCTION

// ---- Objects/Targets/Passive/FB_Wafer.TcPOU
{attribute 'enable_dynamic_creation'}
FUNCTION_BLOCK FB_Wafer EXTENDS FB_TargetBase
VAR_INPUT
END_VAR
VAR_OUTPUT
END_VAR
VAR
	nSquares	: UINT;
END_VAR

METHOD FB_init : BOOL
VAR_INPUT
	bInitRetains : BOOL; // if TRUE, the retain variables are initialized (warm start / cold start)
	bInCopyCode : BOOL;  // if TRUE, the instance afterwards gets moved into the copy code (online change)
END_VAR
eObjectType := E_ObjectType.OBJECTTYPE_Wafer;
eObjectGroup := E_ObjectGroup.OBJECTGROUP_Target;
END_METHOD

METHOD M_AddChild : ERRORID
VAR_INPUT
	pObject : POINTER TO FB_Object;
	nSlotNr	: UINT;
	nIndex 	: INT;
END_VAR
//Kann folgende Objekte aufnehmen:
IF pObject > 0 THEN
	IF pObject^.P_eObjectType = E_ObjectType.OBJECTTYPE_Point OR
		pObject^.P_eObjectType = E_ObjectType.OBJECTTYPE_Slide OR
		pObject^.P_eObjectType = E_ObjectType.OBJECTTYPE_SpotPattern OR
		pObject^.P_eObjectType = E_ObjectType.OBJECTTYPE_SpotArray OR
		pObject^.P_eObjectType = E_ObjectType.OBJECTTYPE_TargetGroup OR
		pObject^.P_eObjectType = E_ObjectType.OBJECTTYPE_Wafer THEN
		M_AddChild := SUPER^.M_AddChild(pObject,nSlotNr,nIndex);
	ELSE
		M_AddChild := E_ErrorIdObjMgmt.ERRORID_InvalidParentObject;
	END_IF
ELSE
	M_AddChild := E_ErrorIdObjMgmt.ERRORID_InvalidParentObject;
END_IF
END_METHOD

METHOD M_GetAllProps : ERRORID
VAR_INPUT
	refCmdData : REFERENCE TO  ST_CmdData;
END_VAR
SUPER^.M_GetAllProps(refCmdData);
nCurrentPropIndex := nCurrentPropIndex + 1;
refCmdData.n32Data[nCurrentPropIndex] := REAL_TO_DINT(rZOffset);
nCurrentPropIndex := nCurrentPropIndex + 1;
refCmdData.n32Data[nCurrentPropIndex] := nSquares;
END_METHOD

METHOD M_SetAllProps : ERRORID
VAR_INPUT
	refCmdData : REFERENCE TO  ST_CmdData;
END_VAR
M_SetAllProps := SUPER^.M_SetAllProps(refCmdData);

IF M_SetAllProps > 0 THEN
	RETURN;
END_IF

nCurrentPropIndex := nCurrentPropIndex + 1;
nSpecPropIndex := nCurrentPropIndex;
rZOffset := DINT_TO_REAL(refCmdData.n32Data[nCurrentPropIndex]);
nCurrentPropIndex := nCurrentPropIndex + 1;
nSquares := DINT_TO_UINT(refCmdData.n32Data[nCurrentPropIndex]);

nNoOfProps := nCurrentPropIndex + 1;
END_METHOD

METHOD M_SetSingleProp : ERRORID
VAR_INPUT
	refCmdData : REFERENCE TO  ST_CmdData;
END_VAR
IF nSpecPropIndex = refCmdData.aHeader[1] THEN
	rZOffset := DINT_TO_REAL(refCmdData.n32Data[0]);
ELSIF (nSpecPropIndex + 1) = refCmdData.aHeader[1] THEN
	nSquares := DINT_TO_UINT(refCmdData.n32Data[0]);
ELSE
	M_SetSingleProp := SUPER^.M_SetSingleProp(refCmdData);
END_IF
END_METHOD

END_FUNCTION_BLOCK
